PROGRAM S_WaferCheckPOU
VAR_INPUT
	bInit				:BOOL:=FALSE;// 初始化状态 busy/done/errDone
	bTrig				:BOOL:=FALSE;// 执行触发 信号
	bReset				:BOOL:=FALSE;// 报错 复位
	bPause				:BOOL:=FALSE;// 暂停 运行
	bStop				:BOOL:=FALSE;// 停止 运行
	bAbort				:BOOL:=FALSE;// 中止 运行
	
END_VAR
VAR_OUTPUT
	busy				:BOOL;
	done				:BOOL;
	errDone				:BOOL;
END_VAR
VAR
	actStep				:ActStepBase;
END_VAR
VAR
	i: INT;
	t1:ton;
	t2:ton;
	t3:ton;
	notchoose:BOOL;
	timeOutTime:TIME:= T#60S;
END_VAR

busy:=actStep.isBusy();
done:=actStep.isDone();
errDone:=actStep.isError();
actStep.Act_Pause(pause:=bPause);

IF bTrig THEN
	bTrig:=FALSE;
	IF NOT busy THEN
		gShowLogTextTitle:='Wafer Check';
		actStep.Act_ex();
	END_IF
END_IF

//状态复位
IF bInit THEN
	bInit:=FALSE;
	Act_init_status();
END_IF

IF bAbort OR bStop THEN
	bAbort:=FALSE;
	bStop:=FALSE;
	Act_init_status();
	actStep.toZeroStep();
	gShowLogTextTitle:='NON';
END_IF
ActionRun(tempActStep:=actStep);

(*
---Trigger action
*)
METHOD Act_Ex : BOOL
VAR_INPUT
END_VAR
IF NOT busy THEN
	actStep.Act_ex();
	Act_Ex:=TRUE;
ELSE
	Act_Ex:=FALSE;
END_IF
END_METHOD

(*
---功能: 状态复位 busy/done/errDone;
*)
METHOD Act_Init_Status
VAR_INPUT
END_VAR
actStep.Act_Init();
END_METHOD

METHOD PRIVATE ActionRun
VAR_INPUT
	tempActStep:ITFActStep;
END_VAR
VAR
END_VAR
VAR_STAT//此处定义静态变量, 保证每次进入该函数时能够在线监控当前值
	tempStep:DINT;
END_VAR
tempStep:=tempActStep.getStep();
CASE tempStep OF
0:
	IF tempActStep.isEx() THEN
		tempActStep.setBusyFlag();
		tempActStep.toBeginStep();
	END_IF
	t1(IN:= FALSE );
	t2(IN:= FALSE );
	t3(IN:= FALSE );
10:
	IF gRunningState<>RunningStatus.eErrorState THEN
		tempActStep.addStep(10,FALSE);
	ELSE
		tempActStep.toErrDoneStep();
	END_IF
20:
	gEnableWaferCheck:=2;
	tempActStep.addStep(10,FALSE);
30:
	IF gEnableWaferCheck=0 THEN// 不检测直接完成
		tempActStep.toStep(100,FALSE);
		t1(IN:= FALSE );
		t2(IN:= FALSE );
		t3(IN:= FALSE );
		RETURN;
	END_IF
	IF gEnableWaferCheck=1 THEN// 检测逻辑
		t1(IN:= FALSE );
		t2(IN:= FALSE );
		t3(IN:= FALSE );
		tempActStep.toStep(100,FALSE);
		RETURN;
	END_IF
	t3(IN:=TRUE,PT:=timeOutTime);
	IF t3.Q THEN
		t1(IN:= FALSE );
		t2(IN:= FALSE );
		t3(IN:= FALSE );
		tempActStep.toErrDoneStep();
		RETURN;
	END_IF
100:
	IF NOT gICP.I_WaferCheck THEN
		tempActStep.addStep(10,FALSE);
	ELSE
		// 机械臂上有晶圆，又需要进行晶圆检测，直接报错
		tempActStep.toErrDoneStep();
	END_IF
110:
	tempActStep.addStep(10,TRUE);
120:
	S_RoughPumping.Act_Init_Status();
	S_RoughPumping.Act_Ex();
	tempActStep.addStep(10,FALSE);
130:
	IF S_RoughPumping.done THEN
		tempActStep.addStep(5,FALSE);
	END_IF
	IF S_RoughPumping.errDone THEN
		tempActStep.toErrDoneStep();
	END_IF	
135:
	IF gEnableWaferCheck=0 THEN// 不检测直接完成
		tempActStep.toDoneStep();
		t1(IN:= FALSE );
		t2(IN:= FALSE );
		t3(IN:= FALSE );
		RETURN;
	END_IF
	IF gEnableWaferCheck=1 THEN// 检测逻辑
		t1(IN:= FALSE );
		t2(IN:= FALSE );
		t3(IN:= FALSE );
		tempActStep.addStep(5,FALSE);
		RETURN;
	END_IF
140:
	IF gICP.PDV.Act_Retract() THEN
		tempActStep.addStep(10,FALSE);
	END_IF
150:
	IF gICP.PDV.Get_Done_Ret() OR gICP.PDVCloseSensor THEN
		tempActStep.addStep(10,FALSE);
	END_IF
160:
	tempActStep.addStep(10,TRUE);
170:
	IF gICP.GateDoorValve.Act_Extend() THEN
		tempActStep.addStep(10,FALSE);
	END_IF
180:
	IF gICP.GateDoorValve.Get_Done_Ext() AND gICP.GateDoorExtSensor THEN
		tempActStep.addStep(10,FALSE);
	END_IF
190:
	tempActStep.addStep(10,TRUE);
200:
	IF NOT gICP.ElectrodeCylRetSensor THEN
		tempActStep.addStep(10,FALSE);
	ELSE
		tempActStep.addStep(30,FALSE);
	END_IF
210:
	tempActStep.addStep(10,TRUE);
220:
	IF gICP.ElectrodeCyl.Act_Retract() THEN
		tempActStep.addStep(10,FALSE);
	END_IF
230:
	IF gICP.ElectrodeCyl.Get_Done_Ret() AND gICP.ElectrodeCylRetSensor THEN
		tempActStep.addStep(10,FALSE);
	END_IF
240:
	tempActStep.addStep(10,TRUE);
250:
	IF gICP.LiftPinCyl.Act_Extend() THEN
		tempActStep.addStep(10,FALSE);
	END_IF
260:
	IF gICP.LiftPinCyl.Get_Done_Ext() AND gICP.LiftPinExtSensor THEN
		tempActStep.addStep(10,FALSE);
	END_IF
270:
	tempActStep.addStep(10,TRUE);
280:
	IF gICP.ARM.Act_HOME_Auto() THEN
		tempActStep.addStep(10,FALSE);
	END_IF
290:
	IF NOT gICP.I_ARMHome THEN// 手臂当前不应该在原点位置
		tempActStep.addStep(10,FALSE);
	END_IF
300:
	t2(IN:=TRUE,PT:=T#10S);
	IF t2.Q AND gICP.ARM.Get_Done_IN() THEN
		t1(IN:= FALSE );
		t2(IN:= FALSE );
		t3(IN:= FALSE );
		tempActStep.toErrDoneStep();
		RETURN;
	END_IF
310:
	tempActStep.addStep(10,TRUE);
320:
	IF gICP.LiftPinCyl.Act_Retract() THEN
		tempActStep.addStep(10,FALSE);
	END_IF
330:
	IF gICP.LiftPinCyl.Get_Done_Ret() AND gICP.LiftPinRetSensor THEN
		tempActStep.addStep(10,FALSE);
	END_IF
340:
	tempActStep.addStep(10,TRUE);
350:
	IF gICP.ARM.Act_HOME_Auto() THEN
		tempActStep.addStep(10,FALSE);
	END_IF
360:
	IF gICP.ARM.Get_Done_HOME() AND gICP.I_ARMHome THEN// 手臂当前不应该在原点位置
		tempActStep.addStep(10,FALSE);
	END_IF
370:
	t2(IN:=TRUE,PT:=T#1S);
	IF t2.Q THEN
		t1(IN:= FALSE );
		t2(IN:= FALSE );
		t3(IN:= FALSE );
		tempActStep.toErrDoneStep();
		RETURN;
	END_IF
380:
	tempActStep.addStep(10,TRUE);
390:
	IF gICP.GateDoorValve.Act_Retract() THEN
		tempActStep.addStep(10,FALSE);
	END_IF
400:
	IF gICP.GateDoorValve.Get_Done_Ret() AND gICP.GateDoorRetSensor THEN
		tempActStep.addStep(10,FALSE);
	END_IF
410:
	IF gICP.I_WaferCheck THEN
		;// wafer记忆状态更新
	ELSE
		;// wafer记忆状态更新
	END_IF
	tempActStep.addStep(10,FALSE);
420:
	tempActStep.toDoneStep();
1000:
	tempActStep.toDoneStep();

60000://Done
	tempActStep.setDoneFlag();
	tempActStep.toZeroStep();
	
65000://Error
	tempActStep.setErrDoneFlag();
	tempActStep.toZeroStep();
END_CASE
END_METHOD

END_PROGRAM

(* stored: Version 1.1.0.1, ProductVersion 3.1.4024.4
   POU S_WaferCheckPOU: Id {93d491af-7e9f-4437-ae6c-10127aa51321}, SpecialFunc None
   Folder Private: Id {b7eb7b00-b8a3-49f0-9335-ea328f543a1c}
   Method Act_Ex: Id {d547058b-8f9b-4b77-8967-de1acf0ac6c4}
   Method Act_Init_Status: Id {0e497cd7-5bfa-423e-9dc7-3ecd96ba88b6}
   Method ActionRun: Id {22ee20cf-a396-424f-a774-29f58cdac048} *)
